// TIA Portal V18 export
FUNCTION "Pallet_NG" : Void   // FC2900, LAD
{ S7_Optimized_Access := 'TRUE' }
// stored: AutoNumber false, SetENOAutomatically false
BEGIN

REGION Network 1
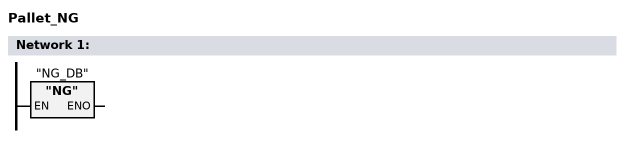
   RUNG wire#powerrail
      "NG_DB"()
   END_RUNG
   // the same network as SCL:
   "NG_DB"();   // "NG"
END_REGION
END_FUNCTION
